Universal Robots PolyScope program: Tool initiation tjeck.urp

Program Tool initiation tjeck (installation=default directory=/programs/usbdisk/Ur-Program/Tool-Initiation createdIn=3.10.1.76190 lastSavedIn=3.10.1.76190 robotSerialNumber=2018359886)
Calibrated DH parameters: a=[-0.000111, -0.180064, -0.391564, 0.000025, 0.000035, 0]; d=[0.089308, 162.079685, -160.155007, -1.814221, 0.094754, 0.082578]; alpha=[1.569707, -0.002379, 0.010338, 1.570474, -1.569894, 0]; deltaTheta=[0.000021, -1.133914, 1.184629, -0.050828, 0.000017, 0.000075]
Robot Program (runOnlyOnce=false)
  Active_tools := 0
  If digital_in[4]≟ False
    old_tool_1 := 1
    Active_tools := Active_tools+1
    SuppressedNode
      Popup Message (haltProgram=false message=Tool 1 active inputType=Text)
  If digital_in[5]≟ False
    old_tool_1 := 2
    Active_tools := Active_tools+1
    SuppressedNode
      Popup Message (haltProgram=false message=Tool 2 active inputType=Text)
  If digital_in[6]≟ False
    old_tool_1 := 3
    Active_tools := Active_tools+1
    SuppressedNode
      Popup Message (haltProgram=false message=Tool 3 active inputType=Text)
  If digital_in[4] and digital_in[5] and digital_in[6]≟ True
    old_tool_1 := 0
    SuppressedNode
      Popup Message (haltProgram=false message=Tool 0 active inputType=Text)
  If Active_tools>1
    Popup Message (haltProgram=false message=Reset Tools inputType=Text)
  SuppressedNode
    Wait Sleep waitTime=5
